Staubli VAL3: ros_server.pjx

--- ros_server.pjx ---
Parameters version=s8.10.3Cs9_BS2093 stackSize=5000 millimeterUnit=true
Program file=dataReceiver.pgx
Program file=dataStreamer.pgx
Program file=decodeMsgBody.pgx
Program file=decodeMsgHeader.pgx
Program file=decTrajPt.pgx
Program file=decTrajPtFull.pgx
Program file=encodeAck.pgx
Program file=encodeJFeedback.pgx
Program file=encodeJState.pgx
Program file=encodeStatus.pgx
Program file=encPrefixHeader.pgx
Program file=encTrajPtAck.pgx
Program file=encTrajPtFAck.pgx
Program file=fetchStatus.pgx
Program file=handleRequest.pgx
Program file=initParams.pgx
Program file=initRosMsgs.pgx
Program file=motionControl.pgx
Program file=motionCtrlVel.pgx
Program file=pushMotion.pgx
Program file=recvData.pgx
Program file=recvHeartbeat.pgx
Program file=recvMsgBody.pgx
Program file=recvMsgHeader.pgx
Program file=recvRosMsg.pgx
Program file=recvTrajPt.pgx
Program file=recvTrajPtFull.pgx
Program file=sendAck.pgx
Program file=sendData.pgx
Program file=sendRosMsg.pgx
Program file=start.pgx
Program file=stateMachine.pgx
Program file=stop.pgx
Program file=toJointArrayRad.pgx
Program file=toJointRxDeg.pgx
Data file=ros_server.dtx
Library alias=IO path=Disk://ros_libs/IOInterface/IOInterface.pjx
Library alias=libQueueFuncs path=Disk://ros_libs/QueueFuncs/QueueFuncs.pjx
Library alias=Staubli path=Disk://ros_libs/Staubli/Staubli.pjx
Library alias=SimpleMsg path=Disk://ros_libs/SimpleMessage/SimpleMessage.pjx
Type name=_MsgRecvState path=Disk://ros_libs/_MsgRecvState/MsgRecvState.pjx
Type name=RosSimpleMsg path=Disk://ros_libs/RosSimpleMsg/RosSimpleMsg.pjx
Type name=RobotStatusMsg path=Disk://ros_libs/RobotStatusMsg/RobotStatusMsg.pjx
Type name=JointStateMsg path=Disk://ros_libs/JointStateMsg/JointStateMsg.pjx
Type name=JointTrajPtMsg path=Disk://ros_libs/JointTrajPtMsg/JointTrajPtMsg.pjx
Type name=JointTrajPtFMsg path=Disk://ros_libs/JointTrajPtFMsg/JointTrajPtFMsg.pjx
Type name=JointFbkMsg path=Disk://ros_libs/JointFbkMsg/JointFbkMsg.pjx
Type name=MotionCmd path=Disk://ros_libs/MotionCmd/MotionCmd.pjx
Type name=Header path=Disk://ros_libs/Header/Header.pjx
Type name=Prefix path=Disk://ros_libs/Prefix/Prefix.pjx
Type name=Body path=Disk://ros_libs/Body/Body.pjx
Type name=Queue path=Disk://ros_libs/Queue/Queue.pjx
Type name=MotionCmdVel path=Disk://ros_libs/MotionCmdVel/MotionCmdVel.pjx
Type name=MotionCfgVel path=Disk://ros_libs/MotionCfgVel/MotionCfgVel.pjx

--- ros_server.dtx ---
public JointFbkMsg rosJointFbkMsg
  [0]
    Body body
      [0]
        num nData[132]
    Header header
      [0]
        num nCommType = 1
        num nData[12]
        num nMsgType = 15
        num nReplyCode
    JointFeedback jointFeedback
      [0]
        num nAccelerations[10]
        num nPositions[10]
        num nRobotId
        num nTime
        num nValidFields
        num nVelocities[10]
    Prefix prefix
      [0]
        num nData[4]
        num nLength = 144
public JointStateMsg rosJointMsg
  [0]
    Body body
      [0]
        num nData[44]
    Header header
      [0]
        num nCommType = 1
        num nData[12]
        num nMsgType = 10
        num nReplyCode
    JointState jointState
      [0]
        num nJoints[10]
        num nSeq
    Prefix prefix
      [0]
        num nData[4]
        num nLength = 56
public JointTrajPtFMsg rosTrajPtFAck
  [0]
    Body body
      [0]
        num nData[136]
    Header header
      [0]
        num nCommType = 3
        num nData[12]
        num nMsgType = 14
        num nReplyCode = 1
    JointTrajPtFull jointTrajPtFull
      [0]
        num nAccelerations[10]
        num nPositions[10]
        num nRobotId
        num nSeq
        num nTime
        num nValidFields
        num nVelocities[10]
    Prefix prefix
      [0]
        num nData[4]
        num nLength = 148
public JointTrajPtFMsg rosTrajPtFMsg
  [0]
    Body body
      [0]
        num nData[136]
    Header header
      [0]
        num nCommType
        num nData[12]
        num nMsgType
        num nReplyCode
    JointTrajPtFull jointTrajPtFull
      [0]
        num nAccelerations[10]
        num nPositions[10]
        num nRobotId
        num nSeq
        num nTime
        num nValidFields
        num nVelocities[10]
    Prefix prefix
      [0]
        num nData[4]
        num nLength = 148
public JointTrajPtMsg rosTrajPtAck
  [0]
    Body body
      [0]
        num nData[52]
    Header header
      [0]
        num nCommType = 3
        num nData[12]
        num nMsgType = 11
        num nReplyCode = 1
    JointTrajPt jointTrajPt
      [0]
        num nDuration
        num nJoints[10]
        num nSeq
        num nVelocity
    Prefix prefix
      [0]
        num nData[4]
        num nLength = 64
public JointTrajPtMsg rosTrajPtMsg
  [0]
    Body body
      [0]
        num nData[52]
    Header header
      [0]
        num nCommType
        num nData[12]
        num nMsgType
        num nReplyCode
    JointTrajPt jointTrajPt
      [0]
        num nDuration
        num nJoints[10]
        num nSeq
        num nVelocity
    Prefix prefix
      [0]
        num nData[4]
        num nLength = 64
MotionCfgVel motionCfgVel
  [0]
    frame fReference = {fatherId=world[0]}
    mdesc mMaxSpeed = {leave=1, reach=1, blend=off}
    num nCmdType
    tool tTool = {fatherId=flange[0], ioLink=valve1}
MotionCmdVel motionCmdVel
  [0]
    num nCmdType
    num nSequence
    num nVelCmd[6]
MotionCmdVel actMotionCmdVel
  [0]
    num nCmdType
    num nSequence
    num nVelCmd[6]
public Queue qMoveBuffer
  [0]
    MotionCmd buffer[10]
      [0]
        jointRx jJointRx
        mdesc mDesc = {leave=0, reach=0}
        num nDuration
        num nSequence
      [1]
        jointRx jJointRx
        mdesc mDesc = {leave=0, reach=0}
        num nDuration
        num nSequence
      [2]
        jointRx jJointRx
        mdesc mDesc = {leave=0, reach=0}
        num nDuration
        num nSequence
      [3]
        jointRx jJointRx
        mdesc mDesc = {leave=0, reach=0}
        num nDuration
        num nSequence
      [4]
        jointRx jJointRx
        mdesc mDesc = {leave=0, reach=0}
        num nDuration
        num nSequence
      [5]
        jointRx jJointRx
        mdesc mDesc = {leave=0, reach=0}
        num nDuration
        num nSequence
      [6]
        jointRx jJointRx
        mdesc mDesc = {leave=0, reach=0}
        num nDuration
        num nSequence
      [7]
        jointRx jJointRx
        mdesc mDesc = {leave=0, reach=0}
        num nDuration
        num nSequence
      [8]
        jointRx jJointRx
        mdesc mDesc = {leave=0, reach=0}
        num nDuration
        num nSequence
      [9]
        jointRx jJointRx
        mdesc mDesc = {leave=0, reach=0}
        num nDuration
        num nSequence
    num nElems
    num nPop
    num nPush
public Queue qTrajPtBuffer
  [0]
    MotionCmd buffer[10]
      [0]
        jointRx jJointRx
        mdesc mDesc = {leave=0, reach=0}
        num nDuration
        num nSequence
      [1]
        jointRx jJointRx
        mdesc mDesc = {leave=0, reach=0}
        num nDuration
        num nSequence
      [2]
        jointRx jJointRx
        mdesc mDesc = {leave=0, reach=0}
        num nDuration
        num nSequence
      [3]
        jointRx jJointRx
        mdesc mDesc = {leave=0, reach=0}
        num nDuration
        num nSequence
      [4]
        jointRx jJointRx
        mdesc mDesc = {leave=0, reach=0}
        num nDuration
        num nSequence
      [5]
        jointRx jJointRx
        mdesc mDesc = {leave=0, reach=0}
        num nDuration
        num nSequence
      [6]
        jointRx jJointRx
        mdesc mDesc = {leave=0, reach=0}
        num nDuration
        num nSequence
      [7]
        jointRx jJointRx
        mdesc mDesc = {leave=0, reach=0}
        num nDuration
        num nSequence
      [8]
        jointRx jJointRx
        mdesc mDesc = {leave=0, reach=0}
        num nDuration
        num nSequence
      [9]
        jointRx jJointRx
        mdesc mDesc = {leave=0, reach=0}
        num nDuration
        num nSequence
    num nElems
    num nPop
    num nPush
public RobotStatusMsg rosStatusMsg
  [0]
    Body body
      [0]
        num nData[28]
    Header header
      [0]
        num nCommType = 1
        num nData[12]
        num nMsgType = 13
        num nReplyCode
    Prefix prefix
      [0]
        num nData[4]
        num nLength = 40
    RobotStatus robotStatus
      [0]
        num nDrivesPowered
        num nEStopped
        num nErrorCode
        num nInError
        num nInMotion
        num nMode
        num nMotionPossible
public RosSimpleMsg genericMotMsg
  [0]
    Header header
      [0]
        num nMsgType
        num nCommType
        num nReplyCode
        num nData[12]
    Prefix prefix
      [0]
        num nLength
        num nData[4]
public RosSimpleMsg genericSysMsg
  [0]
    Header header
      [0]
        num nMsgType
        num nCommType
        num nReplyCode
        num nData[12]
    Prefix prefix
      [0]
        num nLength
        num nData[4]
public RosSimpleMsg genericIOMsg
  [0]
    Header header
      [0]
        num nMsgType
        num nCommType
        num nReplyCode
        num nData[12]
    Prefix prefix
      [0]
        num nLength
        num nData[4]
public _MsgRecvState MsgRecvState
  [0]
    num DECODE_BODY
    num DECODE_HEADER
    num HANDLE_REQUEST
    num PUSH_MOTION
    num RECEIVE_BODY
    num RECEIVE_HEADER
    num SEND_ACK
public bool bDataIn
public bool bDataOut
public bool bDebugMode
public bool bFbkOverrun
public bool bMotionMsgEvent
public bool bMotionOverrun
public bool bOverwriteVel
public bool bRecvOverrun
public bool bScreenOverrun
public bool bShowDebug
public bool bStopNow
public num nConnFlagIO
public num nConnFlagMotion
public num nConnFlagState
public num nConnFlagSystem
public num nDebugCursor
public num nDebugLevel = 5
public num nDebugLevelMax = 7
public num nElapsedTime
public num nHeaderTime = 0.004
num nMotionMode = 1
public num nMotionMsgType
num nMotionPeriod = 0.004
public num nMotionProgress
public num nMoveId = -1
public num nMovePts
public num nPtsPopped
public sio siTcpIpIO = {link=Socket\IO}
public sio siTcpIpMotion = {link=Socket\Motion}
public sio siTcpIpState = {link=Socket\State}
public sio siTcpIpSystem = {link=Socket\System}
public string sHeartbeatTask = "htbtTask"
public string sIORequestTask = "ioRequestTask"
public string sMotionRecvTask = "motionRecvTask"
public string sMotionTask = "motionTask"
public string sScreenTask = "screenTask"
public string sStateMachTask = "stateTask"
public string sStreamerTask = "streamerTask"
public string sSysRequestTask
public tool tTool = {fatherId=flange[0], ioLink=valve1}
jointRx jPosition
jointRx jSpeed

--- start.pgx ---
program start()
  local num l_nFbkPeriod
  local num l_nRecvPeriod
  local num l_nScreenUpdate
begin
  // Copyright (c) 2016, Ocado Technology - Robotics Research Team
  // Copyright (c) 2021, Institute for Factory Automation and Production Systems (FAPS)
  //
  // Licensed under the Apache License, Version 2.0 (the "License");
  // you may not use this file except in compliance with the License.
  // You may obtain a copy of the License at
  //
  //     http://www.apache.org/licenses/LICENSE-2.0
  //
  // Unless required by applicable law or agreed to in writing, software
  // distributed under the License is distributed on an "AS IS" BASIS,
  // WITHOUT WARRANTIES OR CONDITIONS OF ANY KIND, either express or implied.
  // See the License for the specific language governing permissions and
  // limitations under the License.



  // feedback task will run every 4ms (250Hz)
  l_nFbkPeriod=0.004

  // motion control task will run every 4ms (250Hz)
  nMotionPeriod=0.004

  // data (trajectory) reception task will run every 4ms (250Hz)
  l_nRecvPeriod=0.004

  // screen update task will run every 100ms (10Hz)
  l_nScreenUpdate=0.1

  sStreamerTask="streamerTask"
  sMotionRecvTask="motionRecvTask"
  sMotionTask="motionTask"
  sSysRequestTask="sysRequestTask"
  sIORequestTask="ioRequestTask"
  sStateMachTask="stateMachTask"
  sScreenTask="screenTask"
  sHeartbeatTask="htbtTask"

  // initialize TCP/IP parameters and MsgRecvState enum
  call initParams()

  // initialize libraries (must init SimpleMsg first! Staubli is dependent on SimpleMsg)
  call SimpleMsg:init()
  call Staubli:init()
  call IO:init()
  // setup prefix and header of ROS messages
  call initRosMsgs()

  // set standard motion mode
  nMotionMode=Staubli:MotionMode.JOINT_TRAJ

  // socket connection status flags: initially disconnected
  nConnFlagIO = 0
  nConnFlagMotion = 0
  nConnFlagState = 0
  nConnFlagSystem = 0

  // flags defining whether data being received/sent
  bDataIn = false
  bDataOut = false

  // flag defining whether velocity to be overwritten to max. vel.
  bOverwriteVel = false

  nPtsPopped=0
  nMovePts=0

  // flush buffers of sockets
  clearBuffer(siTcpIpIO)
  clearBuffer(siTcpIpMotion)
  clearBuffer(siTcpIpState)
  clearBuffer(siTcpIpSystem)

  // check if robot is not in emergency stop and wait until estop is reset
  if (esStatus() == 2)
    popUpMsg("Please reset E-Stop")
    wait(esStatus() < 2)
  endIf

  // before anything else, enable power (only works if robot is in remote mode)
  if (!isPowered())
    if (workingMode() >= 4)
      do
        enablePower()
        delay(2)
      until isPowered()
    else
      popUpMsg("Power must be enabled manually")
    endIf
  endIf

  // reset motion, potentially setting a start joint position for calling autoConnect() in the future
  resetMotion()

  // create joint state and robot status streamer task to send data to industrial_robot_client
  taskCreateSync sStreamerTask, l_nFbkPeriod, bFbkOverrun, dataStreamer()

  // create receiver task for motion commands (e.g. from industrial_robot_client)
  taskCreateSync sMotionRecvTask, l_nRecvPeriod, bRecvOverrun, dataReceiver(siTcpIpMotion, nConnFlagMotion, genericMotMsg)

  // create motion task to synchronously apply motion commands to robot
  taskCreateSync sMotionTask, nMotionPeriod, bMotionOverrun, motionControl()

  // create asynchronous task to handle state transition
  taskCreate sStateMachTask, 100, stateMachine()

  // create asynchronous task to handle system requests
  taskCreate sSysRequestTask, 100, dataReceiver(siTcpIpSystem, nConnFlagSystem, genericSysMsg)

  // create asynchronous task to handle io requests
  taskCreate sIORequestTask, 100, dataReceiver(siTcpIpIO, nConnFlagIO, genericIOMsg)

  // create asynchronous task to update screen
  //taskCreate sScreenTask, 10, screenUpdate(l_nScreenUpdate)

  // create asynchronous task to receive heartbeat on port 11002
  taskCreate sHeartbeatTask, 10, recvHeartbeat()

end

--- dataReceiver.pgx ---
public program dataReceiver(sio& x_sSocket, num& x_nConnFlag, RosSimpleMsg& x_msg)
  local num l_nMsgRecvState
  local num l_nStartTime
begin
  // Copyright (c) 2016, Ocado Technology - Robotics Research Team
  // Copyright (c) 2021, Institute for Factory Automation and Production Systems (FAPS)
  //
  // Licensed under the Apache License, Version 2.0 (the "License");
  // you may not use this file except in compliance with the License.
  // You may obtain a copy of the License at
  //
  //     http://www.apache.org/licenses/LICENSE-2.0
  //
  // Unless required by applicable law or agreed to in writing, software
  // distributed under the License is distributed on an "AS IS" BASIS,
  // WITHOUT WARRANTIES OR CONDITIONS OF ANY KIND, either express or implied.
  // See the License for the specific language governing permissions and
  // limitations under the License.


  // state machine at initial state
  // 0: RECEIVE_HEADER
  // 1: DECODE_HEADER
  // 2: RECEIVE_BODY
  // 3: DECODE_BODY
  // 4: PUSH_MOTION
  // 5: HANDLE_REQUEST
  // 6: SEND_ACK
  l_nMsgRecvState = MsgRecvState.RECEIVE_HEADER

  while (true)
    // usually for state machines a switch-case statement is a neat implementation
    // HOWEVER, at every iteration of while() this task is sequenced and only called
    // after whatever ms is was defined when created.
    // As a result, receiving one single message, pushing motion and sending ACK
    // would take 6 * task period using switch-case statement.
    // The desirable behaviour is to receive and decode a full message, push motion
    // into buffer and then send ACK to client WITHIN ONE ITERATION of while(),
    // hence the if statement sequence below
    l_nStartTime=clock()

    if (l_nMsgRecvState == MsgRecvState.RECEIVE_HEADER)
      //region @DEBUG
      if (bDebugMode and nDebugLevel<=0)
        //call printDebug("dataReceiver: recvMsgHeader",true)
      endIf
      //endregion

      call recvMsgHeader(x_sSocket,x_nConnFlag,x_msg,l_nMsgRecvState)
    endIf

    nHeaderTime=clock()-l_nStartTime

    if (l_nMsgRecvState == MsgRecvState.DECODE_HEADER)
      //region @DEBUG
      if (bDebugMode and nDebugLevel<=1)
        //call printDebug("dataReceiver: decodeMsgHeader",true)
      endIf
      //endregion

      call decodeMsgHeader(x_msg,l_nMsgRecvState)
    endIf

    if (l_nMsgRecvState == MsgRecvState.RECEIVE_BODY)
      //region @DEBUG
      if (bDebugMode and nDebugLevel<=2)
        //call printDebug("dataReceiver: recvMsgBody",true)
      endIf
      //endregion

      call recvMsgBody(x_sSocket,x_nConnFlag,x_msg,l_nMsgRecvState)
    endIf

    if (l_nMsgRecvState == MsgRecvState.DECODE_BODY)
      //region @DEBUG
      if (bDebugMode and nDebugLevel<=3)
        //call printDebug("dataReceiver: decodeMsgBody",true)
      endIf
      //endregion

      call decodeMsgBody(x_msg,l_nMsgRecvState)
    endIf

    if (l_nMsgRecvState == MsgRecvState.PUSH_MOTION)
      //region @DEBUG
      if (bDebugMode and nDebugLevel<=4)
       //call printDebug("dataReceiver: pushMotion",true)
      endIf
      //endregion

      call pushMotion(x_msg,l_nMsgRecvState)
    endIf

    if (l_nMsgRecvState == MsgRecvState.HANDLE_REQUEST)
      //region @DEBUG
      if (bDebugMode and nDebugLevel<=4)
        //call printDebug("dataReceiver: handleRequest",true)
      endIf
      //endregion

      call handleRequest(x_msg,l_nMsgRecvState)
    endIf

    if (l_nMsgRecvState == MsgRecvState.SEND_ACK)
      //region @DEBUG
      if (bDebugMode and nDebugLevel<=5)
        //call printDebug("dataReceiver: encode/sendAck",true)
      endIf
      //endregion

      call encodeAck(x_msg)
      call sendAck(x_sSocket,x_nConnFlag,x_msg,l_nMsgRecvState)
    endIf

    nElapsedTime=clock()-l_nStartTime-nHeaderTime

    // assert state machine is working OK
    if (l_nMsgRecvState<0 or l_nMsgRecvState>6)
      popUpMsg("Data reception state machine error")
    endIf

    // sequence task
    delay(0)
  endWhile
end

--- dataStreamer.pgx ---
public program dataStreamer()
  local num l_nThrottle
  local num l_nTime
  local num l_nJntSpeed[6]
begin
  // Copyright (c) 2016, Ocado Technology - Robotics Research Team
  // Copyright (c) 2021, Institute for Factory Automation and Production Systems (FAPS)
  //
  // Licensed under the Apache License, Version 2.0 (the "License");
  // you may not use this file except in compliance with the License.
  // You may obtain a copy of the License at
  //
  //     http://www.apache.org/licenses/LICENSE-2.0
  //
  // Unless required by applicable law or agreed to in writing, software
  // distributed under the License is distributed on an "AS IS" BASIS,
  // WITHOUT WARRANTIES OR CONDITIONS OF ANY KIND, either express or implied.
  // See the License for the specific language governing permissions and
  // limitations under the License.



  l_nThrottle = 0
  while (true)
    // only attempt to send data if flag indicates that connection is established
    if (nConnFlagState == 1)
      // fetch current joint feedback data
      l_nTime = clock()
      jPosition = herej()
      $getJntSpeedCmd(l_nJntSpeed)
      jSpeed.j1 = l_nJntSpeed[0]
      jSpeed.j2 = l_nJntSpeed[1]
      jSpeed.j3 = l_nJntSpeed[2]
      jSpeed.j4 = l_nJntSpeed[3]
      jSpeed.j5 = l_nJntSpeed[4]
      jSpeed.j6 = l_nJntSpeed[5]

      // init joint feedback message, valid fields: ( time[0x01] | pos[0x02] | vel[0x04] )
      rosJointFbkMsg.jointFeedback.nRobotId = 0
      rosJointFbkMsg.jointFeedback.nValidFields = 7
      rosJointFbkMsg.jointFeedback.nTime = l_nTime

      // encode and send ROS simple_message ID 15: joint feedback
      call encodeJFeedback(l_nTime, jPosition, jSpeed)
      call sendRosMsg(siTcpIpState, rosJointFbkMsg.prefix, rosJointFbkMsg.header, rosJointFbkMsg.body, nConnFlagState)

      //region @DEBUG
      if (bDebugMode and nDebugLevel==8)
        //call printDebug("dataStreamer: Sent fbk msg", true)
      endIf
      //endregion

      // send Robot Status messages 20 times slower than Joint State
      if (l_nThrottle == 20)
        // fetch robot status
        call fetchStatus()
        // encode and send ROS simple_message ID 13: robot status
        call encodeStatus()
        call sendRosMsg(siTcpIpState, rosStatusMsg.prefix, rosStatusMsg.header, rosStatusMsg.body, nConnFlagState)
        l_nThrottle = 0
      endIf
      l_nThrottle = l_nThrottle + 1
    else
      delay(0.1)
    endIf

    // sequence task
    delay(0)
  endWhile
end

--- decodeMsgBody.pgx ---
public program decodeMsgBody(RosSimpleMsg& x_msg, num& x_nMsgRecvState)
  local bool l_bFlag
begin
  // Copyright (c) 2016, Ocado Technology - Robotics Research Team
  // Copyright (c) 2021, Institute for Factory Automation and Production Systems (FAPS)
  //
  // Licensed under the Apache License, Version 2.0 (the "License");
  // you may not use this file except in compliance with the License.
  // You may obtain a copy of the License at
  //
  //     http://www.apache.org/licenses/LICENSE-2.0
  //
  // Unless required by applicable law or agreed to in writing, software
  // distributed under the License is distributed on an "AS IS" BASIS,
  // WITHOUT WARRANTIES OR CONDITIONS OF ANY KIND, either express or implied.
  // See the License for the specific language governing permissions and
  // limitations under the License.


  // assume failure to decode
  l_bFlag=false

  //region @decode -- call specific decode function
  switch x_msg.header.nMsgType
    case SimpleMsg:MsgType.JOINT_TRAJ_PT
      call decTrajPt(l_bFlag)
    break
    case SimpleMsg:MsgType.JOINT_TRAJ_PT_F
      call decTrajPtFull(l_bFlag)
    break
    // Staubli specific
    case Staubli:MsgType.SET_DRIVE_POWER
      call Staubli:decSetDrvPwrMsg(l_bFlag)
    break
    case Staubli:MsgType.WRITE_SINGLE_IO
      call Staubli:decWriSingIOMsg(l_bFlag)
    break
    case Staubli:MsgType.VELOCITY_CFG
      call Staubli:decodeVelCfg(l_bFlag)
    break
    case Staubli:MsgType.VELOCITY_CMD
      call Staubli:decodeVelCmd(l_bFlag)
    break
    default
      //region @DEBUG
      if (bDebugMode and nDebugLevel<=3)
        //call printDebug("ERROR: unknown msg type ("+toString("",x_msg.header.nMsgType)+")",false)
        //call printDebug("       could not decode message",false)
      endIf
      //endregion
    break
  endSwitch
  //endregion

  //region @check_success -- check whether decoding was successful and move on to the next state
  if (l_bFlag == true)
    switch x_msg.header.nMsgType
      case SimpleMsg:MsgType.JOINT_TRAJ_PT,SimpleMsg:MsgType.JOINT_TRAJ_PT_F,Staubli:MsgType.VELOCITY_CFG,Staubli:MsgType.VELOCITY_CMD
        // move on to state: push motion into buffer
        x_nMsgRecvState = MsgRecvState.PUSH_MOTION
      break
      case Staubli:MsgType.SET_DRIVE_POWER, Staubli:MsgType.WRITE_SINGLE_IO
        // move on to state: handle system/io request
        x_nMsgRecvState = MsgRecvState.HANDLE_REQUEST
      break
    endSwitch

    //region @DEBUG
    if (bDebugMode and nDebugLevel<=3)
      //call printDebug("INFO: decoding successful",false)
    endIf
    //endregion
  else
    // error whilst decoding msg body...
    if (x_msg.header.nCommType==SimpleMsg:CommType.SERVICE_REQUEST)
      // set reply code if comm type is request
      switch x_msg.header.nMsgType
        case SimpleMsg:MsgType.JOINT_TRAJ_PT
          rosTrajPtAck.header.nReplyCode=SimpleMsg:ReplyCode.FAILURE
        break
        case SimpleMsg:MsgType.JOINT_TRAJ_PT_F
          rosTrajPtFAck.header.nReplyCode=SimpleMsg:ReplyCode.FAILURE
        break
        // Staubli specific
        case Staubli:MsgType.SET_DRIVE_POWER
          Staubli:setDrvPwrAck.header.nReplyCode=SimpleMsg:ReplyCode.FAILURE
        break
        case Staubli:MsgType.WRITE_SINGLE_IO
          Staubli:writeSingIOAck.header.nReplyCode=SimpleMsg:ReplyCode.FAILURE
        break
        case Staubli:MsgType.VELOCITY_CFG
          Staubli:velCfgAck.header.nReplyCode=SimpleMsg:ReplyCode.FAILURE
        break
        case Staubli:MsgType.VELOCITY_CMD
          Staubli:velCmdAck.header.nReplyCode=SimpleMsg:ReplyCode.FAILURE
        break
        default
          //region @DEBUG
          if (bDebugMode and nDebugLevel<=3)
            //call printDebug("ERROR: unknown msg type ("+toString("",x_msg.header.nMsgType)+")",false)
            //call printDebug("       could not set reply code",false)
          endIf
          //endregion
        break
      endSwitch
      // jump to state 6: sendAck()
      x_nMsgRecvState = MsgRecvState.SEND_ACK
    else
      // reset state machine, since no ACK is required
      x_nMsgRecvState = MsgRecvState.RECEIVE_HEADER
    endIf
    //region @DEBUG
    if (bDebugMode and nDebugLevel<=3)
      //call printDebug("ERROR: decoding not successful",false)
    endIf
    //endregion
  endIf
  //endregion
end

--- decodeMsgHeader.pgx ---
public program decodeMsgHeader(RosSimpleMsg& x_msg, num& x_nMsgRecvState)
  local num l_nRetVal
begin
  // Copyright (c) 2016, Ocado Technology - Robotics Research Team
  // Copyright (c) 2021, Institute for Factory Automation and Production Systems (FAPS)
  //
  // Licensed under the Apache License, Version 2.0 (the "License");
  // you may not use this file except in compliance with the License.
  // You may obtain a copy of the License at
  //
  //     http://www.apache.org/licenses/LICENSE-2.0
  //
  // Unless required by applicable law or agreed to in writing, software
  // distributed under the License is distributed on an "AS IS" BASIS,
  // WITHOUT WARRANTIES OR CONDITIONS OF ANY KIND, either express or implied.
  // See the License for the specific language governing permissions and
  // limitations under the License.



  // decode message into generic message first
  l_nRetVal=fromBinary(x_msg.prefix.nData,4,"-4l",x_msg.prefix.nLength)
  if (l_nRetVal!=1)
    // error decoding prefix, reset state machine
    x_nMsgRecvState = MsgRecvState.RECEIVE_HEADER
    return
  endIf
  l_nRetVal=fromBinary(x_msg.header.nData,4,"-4l",x_msg.header.nMsgType)
  if (l_nRetVal!=1)
    // error decoding header (msg type), reset state machine
    x_nMsgRecvState = MsgRecvState.RECEIVE_HEADER
    return
  endIf
  l_nRetVal=fromBinary(x_msg.header.nData[4],4,"-4l",x_msg.header.nCommType)
  if (l_nRetVal!=1)
    // error decoding header (comm type), reset state machine
    x_nMsgRecvState = MsgRecvState.RECEIVE_HEADER
    return
  endIf
  l_nRetVal=fromBinary(x_msg.header.nData[8],4,"-4l",x_msg.header.nReplyCode)
  if (l_nRetVal!=1)
    // error decoding header (reply code), reset state machine
    x_nMsgRecvState = MsgRecvState.RECEIVE_HEADER
    return
  endIf

  // no errors detected whilst decoding prefix and header
  // move on to state 2: receive msg body
  x_nMsgRecvState = MsgRecvState.RECEIVE_BODY

  // debug
  if (bDebugMode and nDebugLevel<=1)
    //call printDebug("decodeMsgHeader: successful",true)
    //call printDebug("Prefix    :"+toString("",x_msg.prefix.nLength),false)
    //call printDebug("MsgType   :"+toString("",x_msg.header.nMsgType),false)
    //call printDebug("CommType  :"+toString("",x_msg.header.nCommType),false)
    //call printDebug("ReplyType :"+toString("",x_msg.header.nReplyCode),false)
  endIf
end

--- decTrajPt.pgx ---
public program decTrajPt(bool& x_bFlag)
  local num l_nIndex
  local num l_nRetVal
begin
  // Copyright (c) 2016, Ocado Technology - Robotics Research Team
  //
  // Licensed under the Apache License, Version 2.0 (the "License");
  // you may not use this file except in compliance with the License.
  // You may obtain a copy of the License at
  //
  //     http://www.apache.org/licenses/LICENSE-2.0
  //
  // Unless required by applicable law or agreed to in writing, software
  // distributed under the License is distributed on an "AS IS" BASIS,
  // WITHOUT WARRANTIES OR CONDITIONS OF ANY KIND, either express or implied.
  // See the License for the specific language governing permissions and
  // limitations under the License.



  // decode message ID 11 body (data)

  // assume failure to decode
  rosTrajPtAck.header.nReplyCode=2

  // sequence
  l_nRetVal=fromBinary(rosTrajPtMsg.body.nData,4,"-4l",rosTrajPtMsg.jointTrajPt.nSeq)
  if (l_nRetVal!=1)
    x_bFlag=false
    return
  endIf

  // joints[10]
  for l_nIndex=0 to 9 step 1
    l_nRetVal=fromBinary(rosTrajPtMsg.body.nData[(l_nIndex*4)+4],4,"4.0l",rosTrajPtMsg.jointTrajPt.nJoints[l_nIndex])
    if (l_nRetVal!=1)
      x_bFlag=false
      return
    endIf
  endFor

  // velocity
  l_nRetVal=fromBinary(rosTrajPtMsg.body.nData[44],4,"4.0l",rosTrajPtMsg.jointTrajPt.nVelocity)
  if (l_nRetVal!=1)
    x_bFlag=false
    return
  endIf

  // duration
  l_nRetVal=fromBinary(rosTrajPtMsg.body.nData[48],4,"4.0l",rosTrajPtMsg.jointTrajPt.nDuration)
  if(l_nRetVal!=1)
    x_bFlag=false
    return
  endIf

  // decoding successful
  rosTrajPtAck.header.nReplyCode=1
  rosTrajPtAck.jointTrajPt.nSeq=rosTrajPtMsg.jointTrajPt.nSeq
  nTotalTrajPoint = nTotalTrajPoint + rosTrajPtMsg.jointTrajPt.nSeq+1
  x_bFlag=true
end

--- encodeAck.pgx ---
public program encodeAck(RosSimpleMsg& x_msg)
begin
  // Copyright (c) 2016, Ocado Technology - Robotics Research Team
  // Copyright (c) 2021, Institute for Factory Automation and Production Systems (FAPS)
  //
  // Licensed under the Apache License, Version 2.0 (the "License");
  // you may not use this file except in compliance with the License.
  // You may obtain a copy of the License at
  //
  //     http://www.apache.org/licenses/LICENSE-2.0
  //
  // Unless required by applicable law or agreed to in writing, software
  // distributed under the License is distributed on an "AS IS" BASIS,
  // WITHOUT WARRANTIES OR CONDITIONS OF ANY KIND, either express or implied.
  // See the License for the specific language governing permissions and
  // limitations under the License.



  switch x_msg.header.nMsgType

    case SimpleMsg:MsgType.JOINT_TRAJ_PT
      call encTrajPtAck()
    break

    case SimpleMsg:MsgType.JOINT_TRAJ_PT_F
      call encTrajPtFAck()
    break

    // Staubli specific
    case Staubli:MsgType.SET_DRIVE_POWER
      call Staubli:encSetDrvPwrAck()
    break

    case Staubli:MsgType.WRITE_SINGLE_IO
      call Staubli:encWriSingIOAck()
    break

    case Staubli:MsgType.VELOCITY_CFG
      call Staubli:encodeVelCfgAck()
    break

    case Staubli:MsgType.VELOCITY_CMD
      call Staubli:encodeVelCmdAck()
    break

    default
      //region @DEBUG
      if (bDebugMode and nDebugLevel<=5)
        //call printDebug("encodeAck: switch (msgType)",true)
        //call printDebug("ERROR: unknown msg type",false)
      endIf
      //endregion
    break
  endSwitch
end

--- encodeStatus.pgx ---
public program encodeStatus()
begin
  // Copyright (c) 2016, Ocado Technology - Robotics Research Team
  //
  // Licensed under the Apache License, Version 2.0 (the "License");
  // you may not use this file except in compliance with the License.
  // You may obtain a copy of the License at
  //
  //     http://www.apache.org/licenses/LICENSE-2.0
  //
  // Unless required by applicable law or agreed to in writing, software
  // distributed under the License is distributed on an "AS IS" BASIS,
  // WITHOUT WARRANTIES OR CONDITIONS OF ANY KIND, either express or implied.
  // See the License for the specific language governing permissions and
  // limitations under the License.



  // encode 'prefix' and 'header'
  call encPrefixHeader(rosStatusMsg.prefix, rosStatusMsg.header)

  // encode variables of body message (data)
  toBinary(rosStatusMsg.robotStatus.nDrivesPowered,1,"-4l",rosStatusMsg.body.nData)
  toBinary(rosStatusMsg.robotStatus.nEStopped,1,"-4l",rosStatusMsg.body.nData[4])
  toBinary(rosStatusMsg.robotStatus.nErrorCode,1,"-4l",rosStatusMsg.body.nData[8])
  toBinary(rosStatusMsg.robotStatus.nInError,1,"-4l",rosStatusMsg.body.nData[12])
  toBinary(rosStatusMsg.robotStatus.nInMotion,1,"-4l",rosStatusMsg.body.nData[16])
  toBinary(rosStatusMsg.robotStatus.nMode,1,"-4l",rosStatusMsg.body.nData[20])
  toBinary(rosStatusMsg.robotStatus.nMotionPossible,1,"-4l",rosStatusMsg.body.nData[24])
  toBinary(rosStatusMsg.robotStatus.nTrajectoryComplete,1,"-4l",rosStatusMsg.body.nData[28])
end

--- fetchStatus.pgx ---
public program fetchStatus()
begin
  // Copyright (c) 2016, Ocado Technology - Robotics Research Team
  // Copyright (c) 2021, Institute for Factory Automation and Production Systems (FAPS)
  //
  // Licensed under the Apache License, Version 2.0 (the "License");
  // you may not use this file except in compliance with the License.
  // You may obtain a copy of the License at
  //
  //     http://www.apache.org/licenses/LICENSE-2.0
  //
  // Unless required by applicable law or agreed to in writing, software
  // distributed under the License is distributed on an "AS IS" BASIS,
  // WITHOUT WARRANTIES OR CONDITIONS OF ANY KIND, either express or implied.
  // See the License for the specific language governing permissions and
  // limitations under the License.



  // fetch robot status data

  // drives_powered
  if (isPowered()==true)
    rosStatusMsg.robotStatus.nDrivesPowered=1
  else
    rosStatusMsg.robotStatus.nDrivesPowered=0
  endIf

  // e-stopped
  if (esStatus()==2)
    rosStatusMsg.robotStatus.nEStopped=1
  else
    rosStatusMsg.robotStatus.nEStopped=0
  endIf

  // error_code
  if (taskStatus(sMotionTask) > 1)
    rosStatusMsg.robotStatus.nErrorCode = taskStatus(sMotionTask)
  elseIf (taskStatus(sMotionRecvTask) > 1)
    rosStatusMsg.robotStatus.nErrorCode = taskStatus(sMotionRecvTask)
  elseIf (taskStatus(sStreamerTask) > 1)
    rosStatusMsg.robotStatus.nErrorCode = taskStatus(sStreamerTask)
  elseIf (taskStatus(sHeartbeatTask) > 1)
    rosStatusMsg.robotStatus.nErrorCode = taskStatus(sHeartbeatTask)
  elseIf (taskStatus(sScreenTask) > 1)
    rosStatusMsg.robotStatus.nErrorCode = taskStatus(sScreenTask)
  else
    rosStatusMsg.robotStatus.nErrorCode = 0
  endIf

  // in_error
  if (taskStatus(sMotionRecvTask) == 1 and taskStatus(sMotionTask) == 1 and taskStatus(sStreamerTask) == 1 and taskStatus(sScreenTask) == 1 and taskStatus(sHeartbeatTask) == 1)
    rosStatusMsg.robotStatus.nInError = 0
  else
    rosStatusMsg.robotStatus.nInError = 1
  endIf

  // in_motion
  if (isSettled()==true)
    rosStatusMsg.robotStatus.nInMotion=0
  else
    rosStatusMsg.robotStatus.nInMotion=1
  endIf

  // mode (controller/pendant mode)
  // according to industrial_msgs/RobotMode, possible values are:
  // -1: unknown or unavailable
  //  1: teach or manual mode
  //  2: automatic mode (which I interpret as either local or remote)
  if (workingMode() == 0)
    rosStatusMsg.robotStatus.nMode = -1
  elseIf (workingMode()==1 or workingMode()==2)
    rosStatusMsg.robotStatus.nMode = 1
  elseIf (workingMode()==3 or workingMode()==4)
    rosStatusMsg.robotStatus.nMode = 2
  endIf

  // motion_possible:
  // drives must be powered and e-stop must be off
  // and dataReceiver and motionControl tasks must be
  // running normally
  if(isPowered() == true and esStatus() == 0 and taskStatus(sMotionRecvTask) == 1 and taskStatus(sMotionTask) == 1)
    rosStatusMsg.robotStatus.nMotionPossible=1
  else
    rosStatusMsg.robotStatus.nMotionPossible=0
  endIf

end

--- handleRequest.pgx ---
public program handleRequest(RosSimpleMsg& x_msg, num& x_nMsgRecvState)
  local bool l_bOk
  local num l_nModuleId
  local num l_nPin
  local bool l_bState
begin
  // Copyright (c) 2021, Institute for Factory Automation and Production Systems (FAPS)
  //
  // Licensed under the Apache License, Version 2.0 (the "License");
  // you may not use this file except in compliance with the License.
  // You may obtain a copy of the License at
  //
  //     http://www.apache.org/licenses/LICENSE-2.0
  //
  // Unless required by applicable law or agreed to in writing, software
  // distributed under the License is distributed on an "AS IS" BASIS,
  // WITHOUT WARRANTIES OR CONDITIONS OF ANY KIND, either express or implied.
  // See the License for the specific language governing permissions and
  // limitations under the License.


  // assume success to push motion
  l_bOk=true

  // handle request
  switch x_msg.header.nMsgType
    case Staubli:MsgType.SET_DRIVE_POWER
      if (Staubli:setDrvPwrMsg.bDrivePower==true and isPowered()==false)
        enablePower()
      elseIf (Staubli:setDrvPwrMsg.bDrivePower==false and isPowered()==true)
        disablePower()
      else
        // nothing to do
      endIf
    break
    case Staubli:MsgType.WRITE_SINGLE_IO
      l_nModuleId=Staubli:writeSingIOMsg.writeSingleIO.nModuleId
      l_nPin=Staubli:writeSingIOMsg.writeSingleIO.nPin
      l_bState=Staubli:writeSingIOMsg.writeSingleIO.bState
      call IO:writeSingle(l_nModuleId,l_nPin,l_bState,l_bOk)
    break
    // unknown message type
    default
      l_bOk=false
      //region @DEBUG
      if (bDebugMode and nDebugLevel<=4)
        //call printDebug("ERROR: unknown msg type ("+toString("",x_msg.header.nMsgType)+")",false)
      endIf
      //endregion
    break
  endSwitch

  //region @check_success -- check whether handling request was successful
  if (l_bOk)
    //region @DEBUG
    if (bDebugMode and nDebugLevel<=4)
      //call printDebug("INFO: handling request successful",false)
    endIf
    //endregion
  else
    // could not handle request
    // thus ACK should flag FAILURE, but only if comm type is request
    if (x_msg.header.nCommType==SimpleMsg:CommType.SERVICE_REQUEST)
      switch x_msg.header.nMsgType
        case Staubli:MsgType.SET_DRIVE_POWER
          Staubli:setDrvPwrAck.header.nReplyCode=SimpleMsg:ReplyCode.FAILURE
        break
        case Staubli:MsgType.WRITE_SINGLE_IO
          Staubli:writeSingIOAck.header.nReplyCode=SimpleMsg:ReplyCode.FAILURE
        break
        default
        break
      endSwitch
    endIf
    //region @DEBUG
    if (bDebugMode and nDebugLevel<=4)
      //call printDebug("ERROR: handling request not successful",false)
    endIf
    //endregion
  endIf
  //endregion

  //region @check_reply -- check whether service reply (ACK) should be sent
  if (x_msg.header.nCommType==SimpleMsg:CommType.SERVICE_REQUEST)
    // comm type request requires ACK
    x_nMsgRecvState = MsgRecvState.SEND_ACK
  else
    // other comm types (e.g., topic) does not require ACK, hence skip state
    x_nMsgRecvState = MsgRecvState.RECEIVE_HEADER
  endIf
  //endregion
end

--- initRosMsgs.pgx ---
public program initRosMsgs()
begin
  // Copyright (c) 2016, Ocado Technology - Robotics Research Team
  //
  // Licensed under the Apache License, Version 2.0 (the "License");
  // you may not use this file except in compliance with the License.
  // You may obtain a copy of the License at
  //
  //     http://www.apache.org/licenses/LICENSE-2.0
  //
  // Unless required by applicable law or agreed to in writing, software
  // distributed under the License is distributed on an "AS IS" BASIS,
  // WITHOUT WARRANTIES OR CONDITIONS OF ANY KIND, either express or implied.
  // See the License for the specific language governing permissions and
  // limitations under the License.



  // Joint state message (ID 10)
  // prefix length = 12 + 44
  rosJointMsg.prefix.nLength=56
  rosJointMsg.header.nMsgType=10
  rosJointMsg.header.nCommType=1
  rosJointMsg.header.nReplyCode=0
  // sequence
  rosJointMsg.jointState.nSeq=0



  // Trajectory point message (ID 11)
  // prefix length = 12 + 52
  rosTrajPtAck.prefix.nLength=64
  rosTrajPtAck.header.nMsgType=11
  rosTrajPtAck.header.nCommType=3
  // reply: 1 = success, 2 = failure
  rosTrajPtAck.header.nReplyCode=1
  // joints are assumed to be initiliased to zero

  // the message bellow will be filled upon reception
  rosTrajPtMsg.prefix.nLength=64



  // Robot status message (ID 13)
  // prefix length = 12 + 28
  rosStatusMsg.prefix.nLength=44
  rosStatusMsg.header.nMsgType=13
  rosStatusMsg.header.nCommType=1
  rosStatusMsg.header.nReplyCode=0



  // Trajectory point full message (ID 14)
  // prefix length = 12 + 136
  rosTrajPtFAck.prefix.nLength=148
  rosTrajPtFAck.header.nMsgType=14
  rosTrajPtFAck.header.nCommType=3
  // reply: 1 = success, 2 = failure
  rosTrajPtFAck.header.nReplyCode=1
  // body (data) assumed to be initialised to zero

  // the message bellow will be filled upon reception
  rosTrajPtFMsg.prefix.nLength=148



  // Joint feedback message (ID 15)
  // prefix length = 12 + 132
  rosJointFbkMsg.prefix.nLength=144
  rosJointFbkMsg.header.nMsgType=15
  rosJointFbkMsg.header.nCommType=1
  rosJointFbkMsg.header.nReplyCode=0
end

--- motionControl.pgx ---
public program motionControl()
  local bool l_bFlag
  local bool l_bStopAndClean
  local joint l_jTmp
  local MotionCmd l_mTrajPt
  local MotionCmd l_motion
  local num l_nElems
  local num l_nTime
begin
  // Copyright (c) 2016, Ocado Technology - Robotics Research Team
  // Copyright (c) 2021, Institute for Factory Automation and Production Systems (FAPS)
  //
  // Licensed under the Apache License, Version 2.0 (the "License");
  // you may not use this file except in compliance with the License.
  // You may obtain a copy of the License at
  //
  //     http://www.apache.org/licenses/LICENSE-2.0
  //
  // Unless required by applicable law or agreed to in writing, software
  // distributed under the License is distributed on an "AS IS" BASIS,
  // WITHOUT WARRANTIES OR CONDITIONS OF ANY KIND, either express or implied.
  // See the License for the specific language governing permissions and
  // limitations under the License.



  nMoveId = -1

  while (true)
    // check connection status, and whether to stop motion
    if (nConnFlagMotion == 1 and nConnFlagState == 1 and bStopNow == false)

      // process trajectory point from trajectory buffer
      call libQueueFuncs:getNumElems(qTrajPtBuffer, l_nElems)
      if (l_nElems > 0)
        call libQueueFuncs:pop(qTrajPtBuffer,l_mTrajPt, l_bFlag)
        if (l_bFlag == true)
          nPtsPopped = nPtsPopped + 1
          call libQueueFuncs:push(qMoveBuffer,l_mTrajPt,l_bFlag)
        endIf
      endIf

      // process motion command from move buffer
      // @TODO move buffer should have elements previously interpolated to ensure they are 4 ms apart
      call libQueueFuncs:getNumElems(qMoveBuffer, l_nElems)
      if (l_nElems > 0)
        call libQueueFuncs:pop(qMoveBuffer,l_motion,l_bFlag)
        if (l_bFlag == true)
          nMovePts = nMovePts + 1
          // contrary to what we did earlier, we unconditionally add the traj pt to the motion queue:
          // there doesn't appear to be a way to compare the 'current pose' of the robot to the pts
          // in the trajectory at the appropriate time (ie: when the robot is in motion and about to
          // start executing the segment towards 'l_motion').
          // Checking for dist(l_motion, herej()) (pseudo code) would not be correct as there will
          // always be a delay in the data coming out of herej() and the actual pose of the robot.
          // @TODO potentially set move id according to sequence value
          nMoveId = movej(l_motion.jJointRx, tTool, l_motion.mDesc)

          if (bDebugMode and nDebugLevel<=6)
            l_jTmp=l_motion.jJointRx
            //call printDebug("motionControl: movej() = "+toString("",nMoveId),true)
            //call printDebug("Joint:  "+toString("",l_jTmp.j1)+" "+toString("",l_jTmp.j2)+" "+toString("",l_jTmp.j3)+" "+toString("",l_jTmp.j4)+" "+toString("",l_jTmp.j5)+" "+toString("",l_jTmp.j6),false)
            //call printDebug("vel  :  "+toString("5",l_motion.mDesc.vel),false)
            //call printDebug("tvel :  "+toString("5",l_motion.mDesc.tvel)+"  rvel :  "+toString("5",l_motion.mDesc.rvel),false)
            //call printDebug("accel:  "+toString("5",l_motion.mDesc.accel)+"  decel:  "+toString("5",l_motion.mDesc.decel),false)
          endIf
        endIf
      endIf
    else
      // stop immediately -- resetMotion() also resets moveId
      resetMotion()
      nMoveId = 0

      // clear buffers
      call libQueueFuncs:clear(qTrajPtBuffer)
      call libQueueFuncs:clear(qMoveBuffer)

      // debug
      nPtsPopped = 0
      nMovePts = 0

      // debug
      if (bDebugMode and nDebugLevel==6)
        //call printDebug("motionControl: resetMotion()",true)
        //call printDebug("bStopNow: "+toString("",sel(bStopNow,1,0))+" inConn: "+toString("",nConnFlagMotion)+" outConn: "+toString("",nConnFlagState),false)
      endIf

      // reset stop flag
      bStopNow = false
    endIf

    // store actual move id (progress)
    nMotionProgress = getMoveId()

    // sequence task
    delay(0)
  endWhile
end

--- motionCtrlVel.pgx ---
program motionCtrlVel()
  local bool l_bVelReady
  local num l_nIndex
  local num l_nResult
  local num l_nVelCmd[6]
begin
  // Copyright (c) 2021, Institute for Factory Automation and Production Systems (FAPS)
  //
  // Licensed under the Apache License, Version 2.0 (the "License");
  // you may not use this file except in compliance with the License.
  // You may obtain a copy of the License at
  //
  //     http://www.apache.org/licenses/LICENSE-2.0
  //
  // Unless required by applicable law or agreed to in writing, software
  // distributed under the License is distributed on an "AS IS" BASIS,
  // WITHOUT WARRANTIES OR CONDITIONS OF ANY KIND, either express or implied.
  // See the License for the specific language governing permissions and
  // limitations under the License.


  l_bVelReady=false

  while (true)
    // check connection status and whether to stop motion
    if (nConnFlagMotion==1 and nConnFlagState==1 and bStopNow==false)
      if (l_bVelReady==false)
		// start velocity mode according to configured velocity command type
        switch motionCfgVel.nCmdType
          case Staubli:VelocityType.JOINT
            $velJoint(motionCfgVel.tTool, motionCfgVel.mMaxSpeed)
            l_bVelReady=true
			if (bDebugMode and nDebugLevel==6)
				//call printDebug("motionCtrlVel: $velJoint()",true)
			endIf
          break
          case Staubli:VelocityType.BASE_FRAME
            l_nResult=$velFrame(motionCfgVel.fReference, motionCfgVel.tTool, motionCfgVel.mMaxSpeed)
            if (l_nResult==0)
              l_bVelReady=true
            endIf
			if (bDebugMode and nDebugLevel==6)
				//call printDebug("motionCtrlVel: $velFrame()",true)
				//call printDebug("Result = "+toString("",l_nResult),false)
			endIf
          break
          case Staubli:VelocityType.TOOL_FRAME
            l_nResult=$velTool(motionCfgVel.tTool, motionCfgVel.mMaxSpeed)
            if (l_nResult==0)
              l_bVelReady=true
            endIf
            if (bDebugMode and nDebugLevel==6)
				//call printDebug("motionCtrlVel: $velTool()",true)
				//call printDebug("Result = "+toString("",l_nResult),false)
			endIf
          break
          default
            popUpMsg("Velocity motion command error: Unknown command type ("+toString("",motionCmdVel.nCmdType)+")")
          break
        endSwitch
      endIf

      if (l_bVelReady)
		// - copy global velocity command into local variable for $setVelCmd
		// - store velocity command in other global variable for UI
		// - reset global velocity command (fail-safe, avoiding repeated execution of old commands)
        for l_nIndex=0 to 5
          l_nVelCmd[l_nIndex]=motionCmdVel.nVelCmd[l_nIndex]
          actMotionCmdVel.nVelCmd[l_nIndex]=motionCmdVel.nVelCmd[l_nIndex]
          motionCmdVel.nVelCmd[l_nIndex]=0
        endFor

		// store velocity command type also for displaying in the UI
		actMotionCmdVel.nCmdType=motionCmdVel.nCmdType

        // execute velocity motion command
		$setVelCmd(l_nVelCmd)

        if (bDebugMode and nDebugLevel==6)
          //call printDebug("motionCtrlVel: $setVelCmd()",true)
          //call printDebug("l_nVelCmd = "+toString("",l_nVelCmd[0])+" "+toString("",l_nVelCmd[1])+" "+toString("",l_nVelCmd[2])+" "+toString("",l_nVelCmd[3])+" "+toString("",l_nVelCmd[4])+" "+toString("",l_nVelCmd[5])+" ",false)
        endIf
      endIf
    else
      // stop immediately -- resetMotion() also ends velocity mode
      resetMotion()
      l_bVelReady=false

      // set velocity motion command to initial state
      motionCmdVel.nSequence=0

      for l_nIndex=0 to 5
        motionCmdVel.nVelCmd[l_nIndex]=0
      endFor

      // debug
      if (bDebugMode and nDebugLevel==6)
        //call printDebug("motionCtrlVel: resetMotion()",true)
        //call printDebug("bStopNow: "+toString("",sel(bStopNow,1,0))+" inConn: "+toString("",nConnFlagMotion)+" outConn: "+toString("",nConnFlagState),false)
      endIf

      // reset stop flag
      bStopNow=false
    endIf

    // sequence task
    delay(0)
  endWhile
end

--- pushMotion.pgx ---
public program pushMotion(RosSimpleMsg& x_msg, num& x_nMsgRecvState)
  local bool l_bOk
  local MotionCfgVel l_motCfgVel
  local MotionCmdVel l_motCmdVel
  local MotionCmd l_mTrajPt
  local num l_nConversion
  local num l_nIndex
  local num l_nRad2Deg
begin
  // Copyright (c) 2016, Ocado Technology - Robotics Research Team
  // Copyright (c) 2021, Institute for Factory Automation and Production Systems (FAPS)
  //
  // Licensed under the Apache License, Version 2.0 (the "License");
  // you may not use this file except in compliance with the License.
  // You may obtain a copy of the License at
  //
  //     http://www.apache.org/licenses/LICENSE-2.0
  //
  // Unless required by applicable law or agreed to in writing, software
  // distributed under the License is distributed on an "AS IS" BASIS,
  // WITHOUT WARRANTIES OR CONDITIONS OF ANY KIND, either express or implied.
  // See the License for the specific language governing permissions and
  // limitations under the License.


  l_nRad2Deg = 57.29577951308232

  // assume success to push motion
  l_bOk = true

  if (rosStatusMsg.robotStatus.nMotionPossible == 0)
    // don't push motion into buffer when motion not possible
    l_bOk = false
    // set stop flag so that the motion task resets motion and clears the motion buffers
    bStopNow = true
  endIf

  //region @get_data -- get data from message and store in local variable first
  if (l_bOk)
    switch x_msg.header.nMsgType
      case SimpleMsg:MsgType.JOINT_TRAJ_PT
        l_mTrajPt.nSequence = rosTrajPtMsg.jointTrajPt.nSeq

        // ROS joint position values are in rad, but VAL3 uses degrees
        call toJointRxDeg(rosTrajPtMsg.jointTrajPt.nJoints, l_mTrajPt.jJointRx)

        // from industrial_robot_client/src/joint_trajectory_interface.cpp
        // JointTrajectoryInterface::trajectory_to_msgs()
        // JointTrajectoryInterface::calc_speed()
        // velocity is converted to a scalar value representing % of max velocity,
        // such that 0.2 = 20% of maximum joint speed
      l_mTrajPt.mDesc.vel= limit((rosTrajPtMsg.jointTrajPt.nVelocity * 100), 0, 100)
        l_mTrajPt.nDuration=rosTrajPtMsg.jointTrajPt.nDuration

      break
      case SimpleMsg:MsgType.JOINT_TRAJ_PT_F
        l_mTrajPt.nSequence=rosTrajPtFMsg.jointTrajPtFull.nSeq
        l_mTrajPt.nDuration=rosTrajPtFMsg.jointTrajPtFull.nTime

        // ROS joint position values are in rad, but VAL3 uses degrees
      call toJointRxDeg(rosTrajPtFMsg.jointTrajPtFull.nPositions, l_mTrajPt.jJointRx)

        // from industrial_robot_client/src/joint_trajectory_interface.cpp
        // JointTrajectoryInterface::trajectory_to_msgs()
        // JointTrajectoryInterface::calc_speed()
        // velocity is converted to a scalar value representing % of max velocity,
        // such that 0.2 = 20% of maximum joint speed
      l_mTrajPt.mDesc.vel= limit((rosTrajPtFMsg.jointTrajPtFull.nVelocities[0] * 100), 0, 100)
        // not sure about accelerations as yet
        l_mTrajPt.mDesc.accel=rosTrajPtFMsg.jointTrajPtFull.nAccelerations[0]
        l_mTrajPt.mDesc.decel=l_mTrajPt.mDesc.accel
      break
      // Staubli specific
      case Staubli:MsgType.VELOCITY_CFG
        l_motCfgVel.nCmdType=Staubli:velCfgMsg.velCfg.nCmdType
        link(l_motCfgVel.fReference,world)
        l_motCfgVel.fReference.trsf.x=Staubli:velCfgMsg.velCfg.nRefFrameVec[0]*1000
        l_motCfgVel.fReference.trsf.y=Staubli:velCfgMsg.velCfg.nRefFrameVec[1]*1000
        l_motCfgVel.fReference.trsf.z=Staubli:velCfgMsg.velCfg.nRefFrameVec[2]*1000
        l_motCfgVel.fReference.trsf.rx=Staubli:velCfgMsg.velCfg.nRefFrameVec[3]*l_nRad2Deg
        l_motCfgVel.fReference.trsf.ry=Staubli:velCfgMsg.velCfg.nRefFrameVec[4]*l_nRad2Deg
        l_motCfgVel.fReference.trsf.rz=Staubli:velCfgMsg.velCfg.nRefFrameVec[5]*l_nRad2Deg
        link(l_motCfgVel.tTool,flange)
        l_motCfgVel.tTool.trsf.x=Staubli:velCfgMsg.velCfg.nToolVec[0]*1000
        l_motCfgVel.tTool.trsf.y=Staubli:velCfgMsg.velCfg.nToolVec[1]*1000
        l_motCfgVel.tTool.trsf.z=Staubli:velCfgMsg.velCfg.nToolVec[2]*1000
        l_motCfgVel.tTool.trsf.rx=Staubli:velCfgMsg.velCfg.nToolVec[3]*l_nRad2Deg
        l_motCfgVel.tTool.trsf.ry=Staubli:velCfgMsg.velCfg.nToolVec[4]*l_nRad2Deg
        l_motCfgVel.tTool.trsf.rz=Staubli:velCfgMsg.velCfg.nToolVec[5]*l_nRad2Deg
        l_motCfgVel.mMaxSpeed.accel=limit(Staubli:velCfgMsg.velCfg.nAccel*100,0,100)
        l_motCfgVel.mMaxSpeed.vel=limit(Staubli:velCfgMsg.velCfg.nVel*100,0,100)
        l_motCfgVel.mMaxSpeed.decel=l_motCfgVel.mMaxSpeed.accel
        l_motCfgVel.mMaxSpeed.tvel=Staubli:velCfgMsg.velCfg.nTransVel*1000
        l_motCfgVel.mMaxSpeed.rvel=Staubli:velCfgMsg.velCfg.nRotVel*l_nRad2Deg
      break
      case Staubli:MsgType.VELOCITY_CMD
        l_motCmdVel.nSequence=Staubli:velCmdMsg.velCmd.nSeq
        l_motCmdVel.nCmdType=Staubli:velCmdMsg.velCmd.nCmdType
        if l_motCmdVel.nCmdType==Staubli:VelocityType.JOINT
          for l_nIndex=0 to 5
            l_motCmdVel.nVelCmd[l_nIndex]=Staubli:velCmdMsg.velCmd.nVelVec[l_nIndex]*l_nRad2Deg
          endFor
        elseIf (l_motCmdVel.nCmdType==Staubli:VelocityType.BASE_FRAME) or (l_motCmdVel.nCmdType==Staubli:VelocityType.TOOL_FRAME)
          l_motCmdVel.nVelCmd[0]=Staubli:velCmdMsg.velCmd.nVelVec[0]*1000
          l_motCmdVel.nVelCmd[1]=Staubli:velCmdMsg.velCmd.nVelVec[1]*1000
          l_motCmdVel.nVelCmd[2]=Staubli:velCmdMsg.velCmd.nVelVec[2]*1000
          l_motCmdVel.nVelCmd[3]=Staubli:velCmdMsg.velCmd.nVelVec[3]*l_nRad2Deg
          l_motCmdVel.nVelCmd[4]=Staubli:velCmdMsg.velCmd.nVelVec[4]*l_nRad2Deg
          l_motCmdVel.nVelCmd[5]=Staubli:velCmdMsg.velCmd.nVelVec[5]*l_nRad2Deg
        else
          popUpMsg("Failed to push velocity command. Invalid command type ("+toString("",motionCmdVel.nCmdType)+")")
          for l_nIndex=0 to 5
            l_motCmdVel.nVelCmd[l_nIndex]=0
          endFor
        endIf
      break
      // unknown message type
      default
        l_bOk = false
        //region @DEBUG
        if (bDebugMode and nDebugLevel<=4)
          //call printDebug("ERROR: Unknown msg type ("+toString("",x_msg.header.nMsgType)+")",false)
          //call printDebug("       Failed to get data from msg",false)
        endIf
        //endregion
      break
    endSwitch
    //endregion

    //region @check_special_and_store -- check for special cases before storing motion command
    switch x_msg.header.nMsgType
      case SimpleMsg:MsgType.JOINT_TRAJ_PT,SimpleMsg:MsgType.JOINT_TRAJ_PT_F
        // see github.com/ros-industrial/industrial_core/simple_message/include/simple_message/joint_traj_pt.h
        if (l_mTrajPt.nSequence==-4)
          // set flag to stop immediately
          bStopNow=true
        else
          // check whether velocity value should be overwritten with value set on teach pendant
          if (bOverwriteVel == true)
            // overwrite velocity (and acceleration - ?)
            l_mTrajPt.mDesc.vel = getMonitorSpeed()
            // explicitly setting accel and decel to VAL3 default values
            l_mTrajPt.mDesc.accel = 9999
            l_mTrajPt.mDesc.decel = 9999
          endIf
          // only push motion into buffer if not a STOP message
          // and if joint positions are within software joint limits
          // and if velocity is greater than zero (because movej() will not accept vel <= 0)
          if (isInRange(l_mTrajPt.jJointRx) and l_mTrajPt.mDesc.vel > 0)
            call libQueueFuncs:push(qTrajPtBuffer,l_mTrajPt,l_bOk)
          else
            l_bOk = false
          endIf
          //region @DEBUG
          if (bDebugMode and nDebugLevel<=4)
            //call printDebug("pushMotion: Pushed traj pt",true)
            //call printDebug("bOk: "+toString("",sel(l_bOk,1,0))+" isInRange: "+toString("",sel(isInRange(l_mTrajPt.jJointRx),1,0))+" vel: "+toString("",l_mTrajPt.mDesc.vel),false)
          endIf
          //endregion
        endIf
      break
      // Staubli specific
      case Staubli:MsgType.VELOCITY_CFG
        // @TODO -- check validity of data (e.g. l_motCfgVel.tvel > 0) before storing
        // ... but now only store values in global variable for velocity motion configuration
        motionCfgVel = l_motCfgVel
        //region @DEBUG
        if (bDebugMode and nDebugLevel<=4)
          //call printDebug("pushMotion: Pushed vel cfg", true)
        endIf
        //endregion
      break
      case Staubli:MsgType.VELOCITY_CMD
        // check for special sequence number
        if (l_motCmdVel.nSequence==SimpleMsg:SpecialSeqVal.STOP_TRAJECTORY)
          bStopNow=true
          //region @DEBUG
          if (bDebugMode and nDebugLevel<=4)
            //call printDebug("pushMotion: Stop command!", true)
          endIf
          //endregion
        else
          // @TODO -- probably better to check if (l_motCmdVel.nCmdType == motionCfgVel.nCmdType) to
          //          avoid that the values from l_motCmdVel.nVelCmd are processed with a wrong
          //          reference (joint/frame)
          motionCmdVel = l_motCmdVel
          //region @DEBUG
          if (bDebugMode and nDebugLevel<=4)
            //call printDebug("pushMotion: Pushed vel cmd", true)
          endIf
          //endregion
        endIf
      break
      // unknown message type
      default
        l_bOk=false
        //region @DEBUG
        if (bDebugMode and nDebugLevel<=4)
          //call printDebug("ERROR: Unknown msg type ("+toString("",x_msg.header.nMsgType)+")",false)
          //call printDebug("       Failed to store motion data",false)
        endIf
        //endregion
      break
    endSwitch
  endIf
  //endregion

  //region @check_success -- check whether storing was successful
  if (l_bOk)
    // if successful, setting motion message type and event flag for state machine
    nMotionMsgType = x_msg.header.nMsgType
    switch nMotionMsgType
      case SimpleMsg:MsgType.JOINT_TRAJ_PT, SimpleMsg:MsgType.JOINT_TRAJ_PT_F
        bMotionMsgEvent=true
      break
      case Staubli:MsgType.VELOCITY_CFG
        bMotionMsgEvent = true
      break
      default
        // no state transition required
      break
    endSwitch

    //region @DEBUG
    if (bDebugMode and nDebugLevel<=4)
      if (bMotionMsgEvent)
        //call printDebug("INFO: State transition event ("+toString("",nMotionMsgType)+")",false)
      endIf
    endIf
    //endregion
  else
    // could not push trajectory point into buffer / store motion command
    // thus ACK should flag FAILURE, but only if comm type is request
    if (x_msg.header.nCommType==SimpleMsg:CommType.SERVICE_REQUEST)
      switch x_msg.header.nMsgType
        case SimpleMsg:MsgType.JOINT_TRAJ_PT
          rosTrajPtAck.header.nReplyCode=SimpleMsg:ReplyCode.FAILURE
        break
        case SimpleMsg:MsgType.JOINT_TRAJ_PT_F
          rosTrajPtFAck.header.nReplyCode=SimpleMsg:ReplyCode.FAILURE
        break
        // Staubli specific
        case Staubli:MsgType.VELOCITY_CFG
          Staubli:velCfgAck.header.nReplyCode=SimpleMsg:ReplyCode.FAILURE
        break
        case Staubli:MsgType.VELOCITY_CMD
          Staubli:velCmdAck.header.nReplyCode=SimpleMsg:ReplyCode.FAILURE
        break
        default
        break
      endSwitch
    endIf
    //region @DEBUG
    if (bDebugMode and nDebugLevel<=4)
      //call printDebug("ERROR: Push motion failed",false)
    endIf
    //endregion
  endIf
  //endregion

  //region @check_reply -- check whether service reply (ACK) should be sent
  if (x_msg.header.nCommType == SimpleMsg:CommType.SERVICE_REQUEST)
    // comm type request requires ACK
    x_nMsgRecvState = MsgRecvState.SEND_ACK
  else
    // other comm types (e.g., topic) does not require ACK, hence skip state
    x_nMsgRecvState = MsgRecvState.RECEIVE_HEADER
  endIf
  //endregion
end

--- recvMsgBody.pgx ---
public program recvMsgBody(sio& x_sSocket, num& x_nConnFlag, RosSimpleMsg& x_msg, num& x_nMsgRecvState)
  local bool l_bFlag
begin
  // Copyright (c) 2016, Ocado Technology - Robotics Research Team
  // Copyright (c) 2021, Institute for Factory Automation and Production Systems (FAPS)
  //
  // Licensed under the Apache License, Version 2.0 (the "License");
  // you may not use this file except in compliance with the License.
  // You may obtain a copy of the License at
  //
  //     http://www.apache.org/licenses/LICENSE-2.0
  //
  // Unless required by applicable law or agreed to in writing, software
  // distributed under the License is distributed on an "AS IS" BASIS,
  // WITHOUT WARRANTIES OR CONDITIONS OF ANY KIND, either express or implied.
  // See the License for the specific language governing permissions and
  // limitations under the License.



  l_bFlag=false

  switch x_msg.header.nMsgType
    // standard ROS industrial messages
    case SimpleMsg:MsgType.JOINT_TRAJ_PT
      call recvTrajPt(x_sSocket, x_nConnFlag, x_msg, l_bFlag)
    break
    case SimpleMsg:MsgType.JOINT_TRAJ_PT_F
      call recvTrajPtFull(x_sSocket,x_nConnFlag,x_msg,l_bFlag)
    break
    // Staubli specific
    case Staubli:MsgType.SET_DRIVE_POWER
      call recvRosMsg(x_sSocket, Staubli:setDrvPwrMsg.prefix, Staubli:setDrvPwrMsg.header, Staubli:setDrvPwrMsg.body, x_nConnFlag, x_msg, l_bFlag)
    break
    case Staubli:MsgType.WRITE_SINGLE_IO
      call recvRosMsg(x_sSocket, Staubli:writeSingIOMsg.prefix, Staubli:writeSingIOMsg.header, Staubli:writeSingIOMsg.body, x_nConnFlag, x_msg, l_bFlag)
    break
    case Staubli:MsgType.VELOCITY_CFG
      call recvRosMsg(x_sSocket, Staubli:velCfgMsg.prefix, Staubli:velCfgMsg.header, Staubli:velCfgMsg.body, x_nConnFlag, x_msg, l_bFlag)
    break
    case Staubli:MsgType.VELOCITY_CMD
      call recvRosMsg(x_sSocket, Staubli:velCmdMsg.prefix, Staubli:velCmdMsg.header, Staubli:velCmdMsg.body, x_nConnFlag, x_msg, l_bFlag)
    break
    default
      if (bDebugMode and nDebugLevel<=2)
        //call printDebug("ERROR: unknown msg type ("+toString("",x_msg.header.nMsgType)+")",false)
      endIf
    break
  endSwitch

  if (l_bFlag == true)
    // move on to state 3: decode msg body
    x_nMsgRecvState = MsgRecvState.DECODE_BODY

    // debug
    if (bDebugMode and nDebugLevel<=2)
      //call printDebug("INFO: receiving successful",false)
    endIf
  else
    // error whilst receiving msg body, reset state machine
    x_nMsgRecvState = MsgRecvState.RECEIVE_HEADER
    clearBuffer(x_sSocket)

    // debug
    if (bDebugMode and nDebugLevel<=2)
      //call printDebug("ERROR: receiving not successful",false)
    endIf
  endIf
end

--- sendAck.pgx ---
public program sendAck(sio& x_sSocket, num& x_nConnFlag, RosSimpleMsg& x_msg, num& x_nMsgRecvState)
begin
  // Copyright (c) 2016, Ocado Technology - Robotics Research Team
  // Copyright (c) 2021, Institute for Factory Automation and Production Systems (FAPS)
  //
  // Licensed under the Apache License, Version 2.0 (the "License");
  // you may not use this file except in compliance with the License.
  // You may obtain a copy of the License at
  //
  //     http://www.apache.org/licenses/LICENSE-2.0
  //
  // Unless required by applicable law or agreed to in writing, software
  // distributed under the License is distributed on an "AS IS" BASIS,
  // WITHOUT WARRANTIES OR CONDITIONS OF ANY KIND, either express or implied.
  // See the License for the specific language governing permissions and
  // limitations under the License.



  switch x_msg.header.nMsgType
    case SimpleMsg:MsgType.JOINT_TRAJ_PT
      call sendRosMsg(x_sSocket, rosTrajPtAck.prefix, rosTrajPtAck.header, rosTrajPtAck.body, x_nConnFlag)
    break
    case SimpleMsg:MsgType.JOINT_TRAJ_PT_F
      call sendRosMsg(x_sSocket, rosTrajPtFAck.prefix, rosTrajPtFAck.header, rosTrajPtFAck.body, x_nConnFlag)
    break
    // Staubli specific
    case Staubli:MsgType.SET_DRIVE_POWER
      call sendRosMsg(x_sSocket, Staubli:setDrvPwrAck.prefix, Staubli:setDrvPwrAck.header, Staubli:setDrvPwrAck.body, x_nConnFlag)
    break
    case Staubli:MsgType.WRITE_SINGLE_IO
      call sendRosMsg(x_sSocket, Staubli:writeSingIOAck.prefix, Staubli:writeSingIOAck.header, Staubli:writeSingIOAck.body, x_nConnFlag)
    break
    case Staubli:MsgType.VELOCITY_CFG
      call sendRosMsg(x_sSocket, Staubli:velCfgAck.prefix, Staubli:velCfgAck.header, Staubli:velCfgAck.body, x_nConnFlag)
    break
    case Staubli:MsgType.VELOCITY_CMD
      call sendRosMsg(x_sSocket, Staubli:velCmdAck.prefix, Staubli:velCmdAck.header, Staubli:velCmdAck.body, x_nConnFlag)
    break
    // default
    default
      //region @DEBUG
      if (bDebugMode and nDebugLevel<=5)
        //call printDebug("sendAck: switch (msgType)",true)
        //call printDebug("ERROR: unknown msg type",false)
      endIf
      //endregion
    break
  endSwitch

  // regardless of result from sending ACK
  // reset state machine to receive new messages
  x_nMsgRecvState = MsgRecvState.RECEIVE_HEADER
end

--- stateMachine.pgx ---
program stateMachine()
  local bool l_bKillMotTask
  local bool l_bOk
  local bool l_bResetMotion
  local num l_nNextState
begin
  // Copyright (c) 2021, Institute for Factory Automation and Production Systems (FAPS)
  //
  // Licensed under the Apache License, Version 2.0 (the "License");
  // you may not use this file except in compliance with the License.
  // You may obtain a copy of the License at
  //
  //     http://www.apache.org/licenses/LICENSE-2.0
  //
  // Unless required by applicable law or agreed to in writing, software
  // distributed under the License is distributed on an "AS IS" BASIS,
  // WITHOUT WARRANTIES OR CONDITIONS OF ANY KIND, either express or implied.
  // See the License for the specific language governing permissions and
  // limitations under the License.


  while (true)
    // assume success to state transition
    l_bOk=true
    // reset flags
    l_bKillMotTask=false
    l_bResetMotion=false
    // wait for state transition event
    wait(bMotionMsgEvent)
    bMotionMsgEvent=false

    // //region @DEBUG
    // if (bDebugMode and nDebugLevel==7)
      // call printDebug("stateMachine: got event ("+toString("",nMotionMsgType)+")",true)
      // call printDebug("INFO: current state: "+toString("",nMotionMode),false)
    // endIf
    // //endregion

    //region @switch_current_state -- check whether the current motion task has to be killed
    //                                and set next state
    if (nMotionMode==Staubli:MotionMode.JOINT_TRAJ)

      switch (nMotionMsgType)
        case SimpleMsg:MsgType.JOINT_TRAJ_PT,SimpleMsg:MsgType.JOINT_TRAJ_PT_F
          // already in JOINT_TRAJ mode, skip state transition
          l_bOk=false
        break
        case Staubli:MsgType.VELOCITY_CFG
          l_bKillMotTask=true
          l_nNextState=Staubli:MotionMode.VELOCITY_CTRL
        break
      endSwitch

    elseIf (nMotionMode==Staubli:MotionMode.VELOCITY_CTRL)

      switch (nMotionMsgType)
        case SimpleMsg:MsgType.JOINT_TRAJ_PT,SimpleMsg:MsgType.JOINT_TRAJ_PT_F
          l_bKillMotTask=true
          l_nNextState=Staubli:MotionMode.JOINT_TRAJ
        break
        case Staubli:MsgType.VELOCITY_CFG
          l_bResetMotion=true
        break
      endSwitch

    endIf
    //endregion @switch_current_state

    // check whether to continue
    if (l_bOk)

      //region @DEBUG
      if (bDebugMode and nDebugLevel==7)
        //call printDebug("INFO: state transition ("+toString("",nMotionMode)+" -> "+toString("",l_nNextState)+")",false)
      endIf
      //endregion

      //region @clean_up_motion_task -- if so force motion task to reset motion and/or kill the task
      if (l_bResetMotion)
        // set stop flag (important for velocity mode: reconfiguration without killing task)
        bStopNow=true
      elseIf (l_bKillMotTask)
        // if the current motion task has to be killed, wait until it finishes cleaning up
        bStopNow=true
        wait(bStopNow==false)
        // ... and then kill the task
        taskKill(sMotionTask)
        resetMotion()

        //region @DEBUG
        if (bDebugMode and nDebugLevel==7)
          //call printDebug("INFO: motion task killed",false)
        endIf
        //endregion
      endIf
      //endregion

      //region @create_new_motion_task -- create the new motion task if required
      if (l_bKillMotTask)
        switch l_nNextState
          case Staubli:MotionMode.JOINT_TRAJ
            taskCreateSync sMotionTask,nMotionPeriod,bMotionOverrun,motionControl()
          break
          case Staubli:MotionMode.VELOCITY_CTRL
            taskCreateSync sMotionTask,nMotionPeriod,bMotionOverrun,motionCtrlVel()
          break
          default
            l_bOk=false
            //region @DEBUG
            if (bDebugMode and nDebugLevel==7)
              //call printDebug("ERROR: unknown next state",false)
            endIf
            //endregion
          break
        endSwitch

        //region @DEBUG
        if (bDebugMode and nDebugLevel==7)
          if (l_bOk)
            //call printDebug("INFO: new motion task created",false)
          else
            //call printDebug("ERROR: new motion task not created",false)
          endIf
        endIf
        //endregion
      endIf
      //endregion

      // finally update current state if successful
      if (l_bOk)
        if (l_nNextState!=Staubli:MotionMode.INVALID)
          nMotionMode=l_nNextState

          //region @DEBUG
          if (bDebugMode and nDebugLevel==7)
            //call printDebug("INFO: set new state ("+toString("",l_nNextState)+")",false)
          endIf
          //endregion
        else
          //region @DEBUG
          if (bDebugMode and nDebugLevel==7)
            //call printDebug("WARN: state not set -> invalid ("+toString("",l_nNextState)+")",false)
          endIf
          //endregion
        endIf
      endIf

    endIf

    // sequence task
    delay(0)
  endWhile
end

--- stop.pgx ---
program stop()
begin
  // Copyright (c) 2016, Ocado Technology - Robotics Research Team
  // Copyright (c) 2021, Institute for Factory Automation and Production Systems (FAPS)
  //
  // Licensed under the Apache License, Version 2.0 (the "License");
  // you may not use this file except in compliance with the License.
  // You may obtain a copy of the License at
  //
  //     http://www.apache.org/licenses/LICENSE-2.0
  //
  // Unless required by applicable law or agreed to in writing, software
  // distributed under the License is distributed on an "AS IS" BASIS,
  // WITHOUT WARRANTIES OR CONDITIONS OF ANY KIND, either express or implied.
  // See the License for the specific language governing permissions and
  // limitations under the License.



  resetMotion()
  popUpMsg("Pending movement commands have been cancelled.")
  //userPage(scMonitor)
  //cls(scMonitor)
end
